// TIA Portal project "Scada ile tavan  vinci kontrolü" (V16)

(* hardware
DEVICE "PC-System_1"  SIMATIC PC station
   slot 0: "SIMATIC PC station"  Rail  SIMATIC PC-Station  V1.0
      slot 125: "Stationmanager"  Station_Manager  V6.0.4
   slot 1: "HMI_RT_1"  WinCC RT Professional  6AV2 105-0xxxx-xxxx  16.0.0.0
   slot 2: "IE general_1"  IE General  IE_CP  V8.2.0
DEVICE "S7-1200 station_1"  S7-1200 Station
   slot 0: "Rack_0"  S7-1200 Rack  Rack  V1.0
   slot 1: "PLC_1"  CPU 1214C DC/DC/DC  6ES7 214-1AG40-0XB0  V4.4
*)

// ===== PLC "PLC_1"  CPU 1214C DC/DC/DC =====

VAR_GLOBAL   // PLC tag table "iNPUTS"
   "-X limit sw" AT %I0.0 : Bool;
   "+X limit sw" AT %I0.1 : Bool;
   "+Y limit sw" AT %I0.2 : Bool;
   "-Y limit sw" AT %I0.3 : Bool;
   "-Z limit sw_1" AT %I0.4 : Bool;
   "+Z limit sw_1" AT %I0.5 : Bool;
   "-Z limit sw_2" AT %I0.6 : Bool;
   "+Z limit sw_2" AT %I0.7 : Bool;
   "Termik 1" AT %I1.0 : Bool;
   "Termik 2" AT %I1.1 : Bool;
   "Termik 3" AT %I1.2 : Bool;
   "Termik 4" AT %I1.3 : Bool;
END_VAR

VAR_GLOBAL   // PLC tag table "OUTPUTS"
   "X yön motor ileri" AT %Q0.0 : Bool;
   "X yön motor geri" AT %Q0.1 : Bool;
   "Y yön motor ileri" AT %Q0.2 : Bool;
   "Z yön motor ileri_1" AT %Q0.3 : Bool;
   "Z yön motor ileri_2" AT %Q0.4 : Bool;
   "Z yön motor geri_ 1" AT %Q0.5 : Bool;
   "Z yön motor geri_2" AT %Q0.6 : Bool;
   "Y yön motor geri" AT %Q0.7 : Bool;
END_VAR

DATA_BLOCK "DATALAR"   // DB1
{ S7_Optimized_Access := 'TRUE' }
VERSION : 0.1
   VAR
      "Hmi_Start But" : Bool;
      "Hmi_Stop But" : Bool;
      "Hmi -X yön but" : Bool;
      "Hmi +X  yön but" : Bool;
      "Hmi -Y yön but" : Bool;
      "Hmi +Y yön but" : Bool;
      "Hmi -Z yön but" : Bool;
      "Hmi +Z yön but" : Bool;
      "Sistem genel Start" : Bool;
      "X yön motor lamba" : Bool;
      "Y yön motor lamba" : Bool;
      "Z yön motor  1 lamba" : Bool;
      "Z yön motor  2 lamba" : Bool;
   END_VAR
BEGIN
END_DATA_BLOCK

ORGANIZATION_BLOCK "Main"   // OB1, LAD, ProgramCycle
TITLE = "Main Program Sweep (Cycle)"
{ S7_Optimized_Access := 'TRUE' }
VERSION : 0.1
   VAR_INPUT
      Initial_Call : Bool;   // Initial call of this OB
      Remanence : Bool;   // =True, if remanent data are available
   END_VAR
   VAR_TEMP   // added for the SCL form of the ladder/FBD networks
      _w1 : Bool;
      _w2 : Bool;
   END_VAR
BEGIN

REGION Network 1: SİSTEM GENEL START
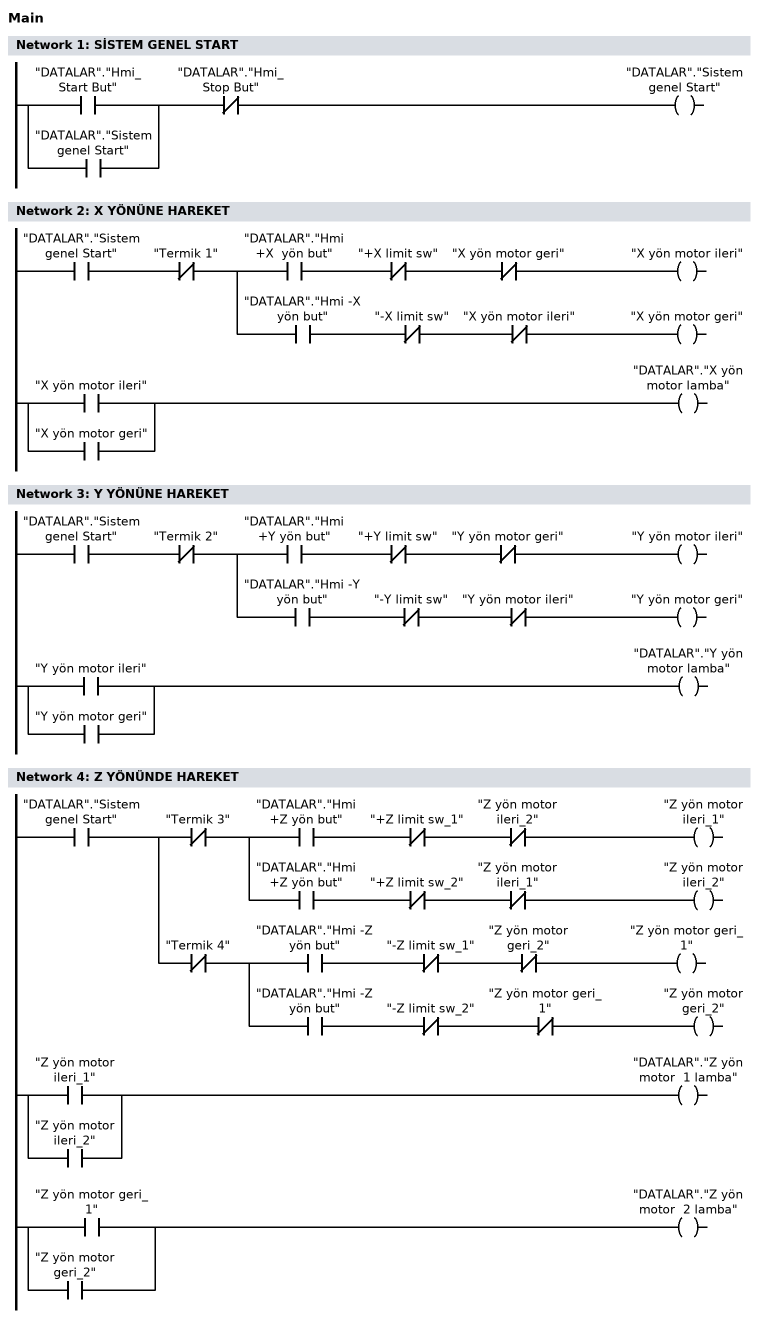
   RUNG wire#powerrail
      Contact( "DATALAR"."Hmi_Start But" )
      wire#w1
      I_Contact( "DATALAR"."Hmi_Stop But" )
      Coil( "DATALAR"."Sistem genel Start" )
   END_RUNG
   RUNG wire#powerrail
      Contact( "DATALAR"."Sistem genel Start" )
   END_RUNG wire#w1
   // the same network as SCL:
   "DATALAR"."Sistem genel Start" := ("DATALAR"."Hmi_Start But" OR "DATALAR"."Sistem genel Start") AND NOT "DATALAR"."Hmi_Stop But";
END_REGION

REGION Network 2: X YÖNÜNE HAREKET
   RUNG wire#powerrail
      Contact( "DATALAR"."Sistem genel Start" )
      I_Contact( "Termik 1" )
      wire#w1
      Contact( "DATALAR"."Hmi +X  yön but" )
      I_Contact( "+X limit sw" )
      I_Contact( "X yön motor geri" )
      Coil( "X yön motor ileri" )
   END_RUNG
   RUNG wire#w1
      Contact( "DATALAR"."Hmi -X yön but" )
      I_Contact( "-X limit sw" )
      I_Contact( "X yön motor ileri" )
      Coil( "X yön motor geri" )
   END_RUNG
   RUNG wire#powerrail
      Contact( "X yön motor ileri" )
      wire#w2
      Coil( "DATALAR"."X yön motor lamba" )
   END_RUNG
   RUNG wire#powerrail
      Contact( "X yön motor geri" )
   END_RUNG wire#w2
   // the same network as SCL:
   #_w1 := "DATALAR"."Sistem genel Start" AND NOT "Termik 1";
   "X yön motor ileri" := #_w1 AND "DATALAR"."Hmi +X  yön but" AND NOT "+X limit sw" AND NOT "X yön motor geri";
   "X yön motor geri" := #_w1 AND "DATALAR"."Hmi -X yön but" AND NOT "-X limit sw" AND NOT "X yön motor ileri";
   "DATALAR"."X yön motor lamba" := "X yön motor ileri" OR "X yön motor geri";
END_REGION

REGION Network 3: Y YÖNÜNE HAREKET
   RUNG wire#powerrail
      Contact( "DATALAR"."Sistem genel Start" )
      I_Contact( "Termik 2" )
      wire#w1
      Contact( "DATALAR"."Hmi +Y yön but" )
      I_Contact( "+Y limit sw" )
      I_Contact( "Y yön motor geri" )
      Coil( "Y yön motor ileri" )
   END_RUNG
   RUNG wire#w1
      Contact( "DATALAR"."Hmi -Y yön but" )
      I_Contact( "-Y limit sw" )
      I_Contact( "Y yön motor ileri" )
      Coil( "Y yön motor geri" )
   END_RUNG
   RUNG wire#powerrail
      Contact( "Y yön motor ileri" )
      wire#w2
      Coil( "DATALAR"."Y yön motor lamba" )
   END_RUNG
   RUNG wire#powerrail
      Contact( "Y yön motor geri" )
   END_RUNG wire#w2
   // the same network as SCL:
   #_w1 := "DATALAR"."Sistem genel Start" AND NOT "Termik 2";
   "Y yön motor ileri" := #_w1 AND "DATALAR"."Hmi +Y yön but" AND NOT "+Y limit sw" AND NOT "Y yön motor geri";
   "Y yön motor geri" := #_w1 AND "DATALAR"."Hmi -Y yön but" AND NOT "-Y limit sw" AND NOT "Y yön motor ileri";
   "DATALAR"."Y yön motor lamba" := "Y yön motor ileri" OR "Y yön motor geri";
END_REGION

REGION Network 4: Z YÖNÜNDE HAREKET
   RUNG wire#powerrail
      Contact( "DATALAR"."Sistem genel Start" )
      wire#w1
      I_Contact( "Termik 3" )
      wire#w2
      Contact( "DATALAR"."Hmi +Z yön but" )
      I_Contact( "+Z limit sw_1" )
      I_Contact( "Z yön motor ileri_2" )
      Coil( "Z yön motor ileri_1" )
   END_RUNG
   RUNG wire#w2
      Contact( "DATALAR"."Hmi +Z yön but" )
      I_Contact( "+Z limit sw_2" )
      I_Contact( "Z yön motor ileri_1" )
      Coil( "Z yön motor ileri_2" )
   END_RUNG
   RUNG wire#w1
      I_Contact( "Termik 4" )
      wire#w3
      Contact( "DATALAR"."Hmi -Z yön but" )
      I_Contact( "-Z limit sw_1" )
      I_Contact( "Z yön motor geri_2" )
      Coil( "Z yön motor geri_ 1" )
   END_RUNG
   RUNG wire#w3
      Contact( "DATALAR"."Hmi -Z yön but" )
      I_Contact( "-Z limit sw_2" )
      I_Contact( "Z yön motor geri_ 1" )
      Coil( "Z yön motor geri_2" )
   END_RUNG
   RUNG wire#powerrail
      Contact( "Z yön motor ileri_1" )
      wire#w4
      Coil( "DATALAR"."Z yön motor  1 lamba" )
   END_RUNG
   RUNG wire#powerrail
      Contact( "Z yön motor ileri_2" )
   END_RUNG wire#w4
   RUNG wire#powerrail
      Contact( "Z yön motor geri_ 1" )
      wire#w5
      Coil( "DATALAR"."Z yön motor  2 lamba" )
   END_RUNG
   RUNG wire#powerrail
      Contact( "Z yön motor geri_2" )
   END_RUNG wire#w5
   // the same network as SCL:
   #_w1 := "DATALAR"."Sistem genel Start" AND NOT "Termik 3";
   "Z yön motor ileri_1" := #_w1 AND "DATALAR"."Hmi +Z yön but" AND NOT "+Z limit sw_1" AND NOT "Z yön motor ileri_2";
   "Z yön motor ileri_2" := #_w1 AND "DATALAR"."Hmi +Z yön but" AND NOT "+Z limit sw_2" AND NOT "Z yön motor ileri_1";
   #_w2 := "DATALAR"."Sistem genel Start" AND NOT "Termik 4";
   "Z yön motor geri_ 1" := #_w2 AND "DATALAR"."Hmi -Z yön but" AND NOT "-Z limit sw_1" AND NOT "Z yön motor geri_2";
   "Z yön motor geri_2" := #_w2 AND "DATALAR"."Hmi -Z yön but" AND NOT "-Z limit sw_2" AND NOT "Z yön motor geri_ 1";
   "DATALAR"."Z yön motor  1 lamba" := "Z yön motor ileri_1" OR "Z yön motor ileri_2";
   "DATALAR"."Z yön motor  2 lamba" := "Z yön motor geri_ 1" OR "Z yön motor geri_2";
END_REGION
END_ORGANIZATION_BLOCK

(* ===== HMI "HMI_RT_1" =====
system functions are stored by id; their names below are inferred from use
connection "HMI_Connection_1": S71200_TCP_IP, SCADA_S7_1200

HMI tags "Default tag table"
   "1" : Bool = PLC 1 AT %I0.0, 500 ms
   "DATALAR_Hmi_StartBut" : Bool = PLC DATALAR."Hmi_Start But", 500 ms
   "DATALAR_Hmi_StopBut" : Bool = PLC DATALAR."Hmi_Stop But", 500 ms
   "DATALAR_Hmi+Xyönbut" : Bool = PLC DATALAR."Hmi +X  yön but", 500 ms
   "DATALAR_Hmi-Xyönbut" : Bool = PLC DATALAR."Hmi -X yön but", 500 ms
   "DATALAR_Hmi-Yyönbut" : Bool = PLC DATALAR."Hmi -Y yön but", 500 ms
   "DATALAR_Hmi+Zyönbut" : Bool = PLC DATALAR."Hmi +Z yön but", 500 ms
   "DATALAR_Hmi+Yyönbut" : Bool = PLC DATALAR."Hmi +Y yön but", 500 ms
   "DATALAR_Hmi-Zyönbut" : Bool = PLC DATALAR."Hmi -Z yön but", 500 ms
   "DATALAR_Zyönmotor1lamba" : Bool = PLC DATALAR."Z yön motor  1 lamba", 500 ms
   "DATALAR_Zyönmotor2lamba" : Bool = PLC DATALAR."Z yön motor  2 lamba", 500 ms
   "DATALAR_Yyönmotorlamba" : Bool = PLC DATALAR."Y yön motor lamba", 500 ms
   "DATALAR_Xyönmotorlamba" : Bool = PLC DATALAR."X yön motor lamba", 500 ms
   "Xyönmotorileri" : Bool = PLC "X yön motor ileri" AT %Q0.0, 500 ms
   "Xyönmotorgeri" : Bool = PLC "X yön motor geri" AT %Q0.1, 500 ms
   "Yyönmotorgeri" : Bool = PLC "Y yön motor geri" AT %Q0.7, 500 ms
   "Yyönmotorileri" : Bool = PLC "Y yön motor ileri" AT %Q0.2, 500 ms
   "Zyönmotorileri_1" : Bool = PLC "Z yön motor ileri_1" AT %Q0.3, 500 ms
   "Zyönmotorileri_2" : Bool = PLC "Z yön motor ileri_2" AT %Q0.4, 500 ms

screen "ANA SAYFA" 1024x768
   TextField "Text field_1" at 251,19 size 427x43; Text 'Tava Vinci Kontrolü Ekranı'
   GraphicView "Graphic view_1" at 81,94 size 726x486; Picture "crane-1024x576"
   Button "Button_1" at 838,209 size 150x85; TextOff 'START BUT'
      on PressLeft: SetBit("DATALAR_Hmi_StartBut")
      on ReleaseLeft: ResetBit("DATALAR_Hmi_StartBut")
      Appearance <- "DATALAR_Hmi_StartBut"
   Button "Button_2" at 839,322 size 151x82; TextOff 'STOP BUT'
      on PressLeft: SetBit("DATALAR_Hmi_StopBut")
      on ReleaseLeft: ResetBit("DATALAR_Hmi_StopBut")
      Appearance <- "DATALAR_Hmi_StopBut"
   Circle "Circle_1" at 650,303 size 24x24
      Appearance <- "DATALAR_Zyönmotor1lamba"
   Circle "Circle_2" at 411,400 size 21x21
      Appearance <- "DATALAR_Zyönmotor2lamba"
   Circle "Circle_3" at 384,155 size 20x20
      Appearance <- "DATALAR_Xyönmotorlamba"
   Circle "Circle_4" at 523,215 size 21x21
      Appearance <- "DATALAR_Yyönmotorlamba"
   Button "Button_3" at 69,527 size 181x46; TextOff '-X YÖNĞNE GİT'
      on PressLeft: SetBit("DATALAR_Hmi+Xyönbut")
      on ReleaseLeft: ResetBit("DATALAR_Hmi+Xyönbut")
      Appearance <- "DATALAR_Hmi+Xyönbut"
   Button "Button_4" at 69,582 size 181x46; TextOff '+X YÖNĞNE GİT'
      on PressLeft: SetBit("DATALAR_Hmi-Xyönbut")
      on ReleaseLeft: ResetBit("DATALAR_Hmi-Xyönbut")
      Appearance <- "DATALAR_Hmi-Xyönbut"
   Button "Button_5" at 277,525 size 181x46; TextOff '-Y YÖNĞNE GİT'
      on PressLeft: SetBit("DATALAR_Hmi-Yyönbut")
      on ReleaseLeft: ResetBit("DATALAR_Hmi-Yyönbut")
      Appearance <- "DATALAR_Hmi-Yyönbut"
   Button "Button_6" at 280,580 size 181x46; TextOff '+Y YÖNĞNE GİT'
      on PressLeft: SetBit("DATALAR_Hmi+Yyönbut")
      on ReleaseLeft: ResetBit("DATALAR_Hmi+Yyönbut")
   Button "Button_7" at 496,525 size 181x46; TextOff '-Z YÖNĞNE GİT'
      on PressLeft: SetBit("DATALAR_Hmi-Zyönbut")
      on ReleaseLeft: ResetBit("DATALAR_Hmi-Zyönbut")
      Appearance <- "DATALAR_Hmi-Zyönbut"
   Button "Button_8" at 497,581 size 181x46; TextOff '+Z YÖNĞNE GİT'
      on PressLeft: SetBit("DATALAR_Hmi+Zyönbut")
      on ReleaseLeft: ResetBit("DATALAR_Hmi+Zyönbut")
      Appearance <- "DATALAR_Hmi+Zyönbut"
   TextField "Text field_2" at 755,572 size 227x23; Text 'VİNÇ -Y YÖNÜNE GİDİYOR'
      Visibility <- "Yyönmotorgeri"
   TextField "Text field_3" at 756,510 size 227x23; Text 'VİNÇ -X YÖNÜNE GİDİYOR'
      Visibility <- "Xyönmotorileri"
   TextField "Text field_4" at 758,540 size 203x19; Text 'VİNÇ +X YÖNÜNE GİDİYOR'
      Visibility <- "Xyönmotorgeri"
   TextField "Text field_5" at 754,605 size 204x19; Text 'VİNÇ +Y YÖNÜNE GİDİYOR'
      Visibility <- "Yyönmotorileri"
   TextField "Text field_6" at 753,633 size 234x23; Text 'VİNÇ +Z YÖNÜNE GİDİYOR'
      Visibility <- "Zyönmotorileri_1"
   TextField "Text field_7" at 754,663 size 227x23; Text 'VİNÇ -Z YÖNÜNE GİDİYOR'
      Visibility <- "Zyönmotorileri_2"
*)